{attribute 'linkalways'} 
{attribute 'no_explicit_call' := 'This FB is a CLASS and must be accessed using methods or properties'}
{attribute 'enable_dynamic_creation'}
FUNCTION_BLOCK _ETcVnColorMapSize EXTENDS EnumDatatypeBase
VAR
	localData : ETcVnColorMapSize;
	activeData : REFERENCE TO ETcVnColorMapSize;
	enumBaseDatatype : _UDINT(localData);
END_VAR

METHOD PRIVATE AddLocalEnumeration
VAR_INPUT
	Enumeration : T_MAXSTRING;
	Value : ETcVnColorMapSize;
END_VAR
AddEnumeration(Enumeration, Value);
END_METHOD

PROPERTY PUBLIC Address : PVOID
GET
Address := ADR(activeData);
END_GET
END_PROPERTY

METHOD PUBLIC ClearReference
VAR_INPUT
END_VAR
activeData REF= localData;
SetBaseDatatypeReference();
END_METHOD

METHOD PUBLIC Clone : I_Datatype
VAR
    pClone : POINTER TO _ETcVnColorMapSize;
END_VAR
pClone := __NEW(_ETcVnColorMapSize(InitialValue := Value));
Clone := pClone^;
END_METHOD

METHOD FB_init : BOOL
VAR_INPUT
	bInitRetains : BOOL; // if TRUE, the retain variables are initialized (warm start / cold start)
	bInCopyCode : BOOL;  // if TRUE, the instance afterwards gets moved into the copy code (online change)
	InitialValue : ETcVnColorMapSize;
END_VAR
localData := InitialValue;
AddBaseDatatype(enumBaseDatatype);
ClearReference();

AddLocalEnumeration('TCVN_CMS_256', ETcVnColorMapSize.TCVN_CMS_256);
AddLocalEnumeration('TCVN_CMS_65536', ETcVnColorMapSize.TCVN_CMS_65536);
END_METHOD

PROPERTY PUBLIC Identifier : T_MAXSTRING
GET
Identifier := 'ETcVnColorMapSize';
END_GET
END_PROPERTY

METHOD IsEnumeratorValueEqual : BOOL
VAR_INPUT
	Enumerator : I_KeyValueForwardEnumerator;
END_VAR
VAR
	storedValue : ETcVnColorMapSize;
END_VAR
IF NOT Enumerator.TryGet(storedValue) THEN
	RETURN;
END_IF

IsEnumeratorValueEqual := storedValue = activeData;
END_METHOD

METHOD PUBLIC MakeReferenceTo
VAR_INPUT
	ReferenceTarget : REFERENCE TO ETcVnColorMapSize;
END_VAR
activeData REF= ReferenceTarget;
SetBaseDatatypeReference();
END_METHOD

METHOD PROTECTED SetBaseDatatypeReference
VAR_INPUT
END_VAR
enumBaseDatatype.MakeReferenceTo(activeData);
END_METHOD

PROPERTY PUBLIC Size : UDINT
GET
Size := SIZEOF(activeData);
END_GET
END_PROPERTY

METHOD TryMakeReferenceTo : BOOL
VAR_INPUT
	Target : I_Datatype;
END_VAR
VAR
	pTargetData : POINTER TO ETcVnColorMapSize;
END_VAR
IF NOT IsEquivalentTo(Target) THEN
	RETURN;
END_IF

pTargetData := Target.Address;
activeData REF= pTargetData^;
SetBaseDatatypeReference();
TryMakeReferenceTo := TRUE;
END_METHOD

PROPERTY PUBLIC Value : ETcVnColorMapSize
GET
Value := activeData;
END_GET
SET
activeData := Value;
END_SET
END_PROPERTY

END_FUNCTION_BLOCK

(* stored: Version 1.1.0.1, ProductVersion 3.1.4024.13
   POU _ETcVnColorMapSize: Id {a5fb792c-17bb-42c1-b662-ccf221c7b18f}, SpecialFunc None
   Folder Core: Id {27b1847f-72a4-0adc-0985-2dc3b12e2f83}
   Folder Protected: Id {916c6c11-e204-0d1c-2030-5e39bfe3c98c}
   Folder Customize: Id {0746a25e-89bf-0990-1a1f-e8e4f743d33b}
   Folder Constructor: Id {22d4d79b-cf1a-4956-9910-9590b91ecc15}
   Folder Private: Id {ac421bb5-33f5-4c40-bfb3-9d2f25fca1e7}
   Folder Protected: Id {e658752b-183d-4a33-8be1-e89327c6fb45}
   Method AddLocalEnumeration: Id {51a24347-b85b-406c-9186-b929ba8c06f0}
   Property Address: Id {c8b3c879-6ea7-0784-248b-c0874e23282d}
   Get Get: Id {4fd78abd-5db7-0a0e-0378-032d71b35b1f}
   Method ClearReference: Id {a112063e-36fb-06c9-19ac-b2c12eb69687}
   Method Clone: Id {ab435455-8572-47e7-a6b6-c833c0fefc0d}
   Method FB_init: Id {dd3858e0-9762-4633-808b-ec69f4c9045c}
   Property Identifier: Id {314ce15b-3e09-42e3-b896-e42819d9820a}
   Get Get: Id {40b53494-0f44-48d1-8a44-efb1c8aa6e75}
   Method IsEnumeratorValueEqual: Id {2d5962b0-5a23-4e53-b303-fc9ca768646b}
   Method MakeReferenceTo: Id {c5983ada-e994-42f0-b6a2-ec52aa03f706}
   Method SetBaseDatatypeReference: Id {661ab6c0-f225-03eb-0e83-c35e3e7a8b7b}
   Property Size: Id {4561ed51-63d0-0b21-0b88-e0ada96d0d23}
   Get Get: Id {6d0467e9-ad21-0288-0754-c704acfccd3a}
   Method TryMakeReferenceTo: Id {13b1f4b6-d568-47d3-996e-2ec8d8ef7bfe}
   Property Value: Id {58a8e867-3b6b-4ec7-834a-cd5fc0eb2366}
   Get Get: Id {08c9002d-086e-41ee-9b43-8232930cc733}
   Set Set: Id {5f92f431-13b0-4821-8d8e-aa575a2b785a} *)
